{attribute 'qualified_only'}
{attribute 'strict'}
{attribute 'to_string'}
TYPE enErrorBitNumber :
(
	Pressure := 0,
	Flame:=1,
	BurnerTemperature:=2
);
END_TYPE

(* stored: Version 1.1.0.1
   DUT enErrorBitNumber: Id {adbd0c05-dc60-4564-9827-25c3e558ff96} *)
